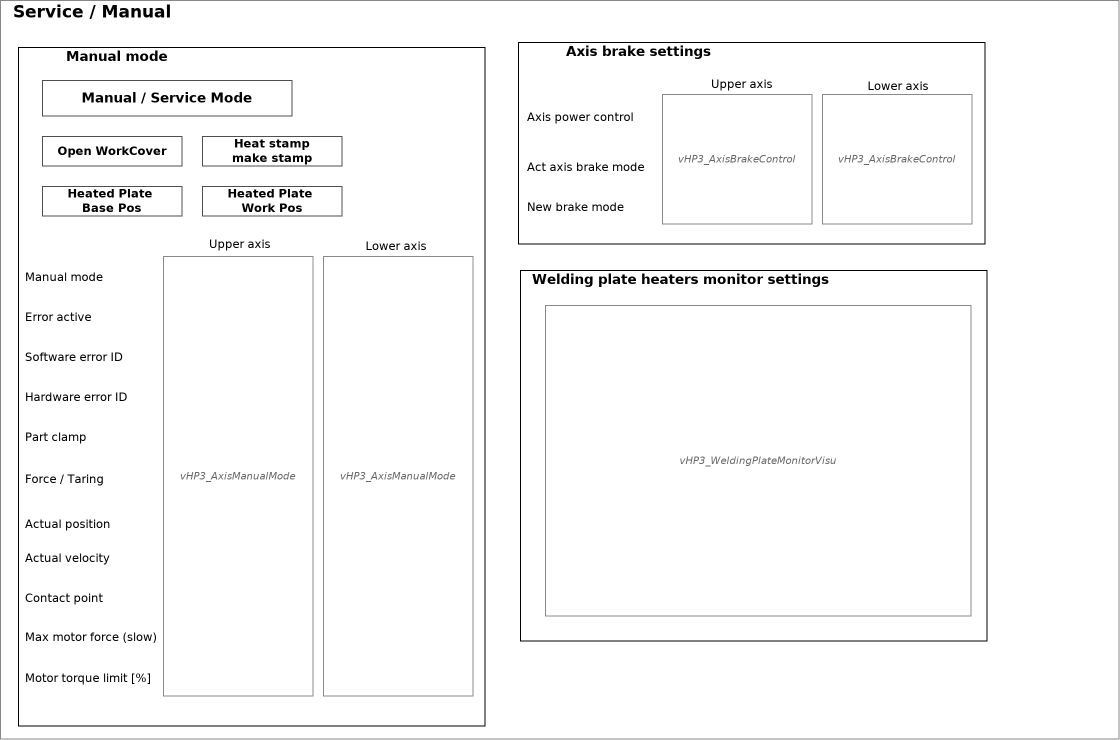
VISUALIZATION vHP3_MachineSub_Service  // 1120x740
VAR_IN_OUT
	fbHP: fbHPv3_Control;
END_VAR
    RoundedRectangle (18,47 467x679), "Manual mode"
    Rectangle (42,80 250x36), "Manual / Service Mode", colour toggle: fbHP.bManualMode
        toggle fbHP.bManualMode
    Label (22,265 130x24), "Manual mode"
    Label (22,512 130x24), "Actual position"
    Label (22,546 130x24), "Actual velocity"
    Label (22,625 145x24), "Max motor force (slow)"
    Rectangle (42,136 140x30), "Open WorkCover", colour toggle: fbHP.bWorkCover_Riseup, input disabled if: NOT fbHP.bManualMode
        toggle fbHP.bWorkCover_Riseup p2164770859=TRUE
    Rectangle (42,186 140x30), "Heated Plate Base Pos", colour toggle: fbHP.fbHeatedPlate_Actuator.Closed, input disabled if: NOT fbHP.bManualMode
        OnMouseClick: execute { fbHP.fbHeatedPlate_Actuator.mClose(); }
    Rectangle (202,186 140x30), "Heated Plate Work Pos", colour toggle: fbHP.fbHeatedPlate_Actuator.Opened, input disabled if: NOT fbHP.bManualMode
        OnMouseClick: execute { fbHP.fbHeatedPlate_Actuator.mOpen(); }
    Rectangle (202,136 140x30), "Heat stamp make stamp", colour toggle: fbHP.bMakeStamp, invisible if: NOT fbHP.bMarkingAsembled, input disabled if: NOT fbHP.bManualMode
        toggle fbHP.bMakeStamp
        OnMouseClick: execute { fbHP.fbHeatedPlate_Actuator.mClose(); }
    Label (175,232 130x24), "Upper axis"
    Label (331,234 130x24), "Lower axis"
    Label (22,666 145x24), "Motor torque limit [%]"
    RoundedRectangle (10,0 300x26), "Service / Manual"
    Frame (163,256 150x440)
        shows vHP3_AxisManualMode(fbData := fbHP.fbAxisUp)
    Frame (323,256 150x440)
        shows vHP3_AxisManualMode(fbData := fbHP.fbAxisDn)
    Label (22,305 130x24), "Error active"
    Label (22,345 130x24), "Software error ID"
    Label (22,385 130x24), "Hardware error ID"
    Label (22,467 130x24), "Force / Taring"
    Label (22,425 130x24), "Part clamp"
    Label (22,586 130x24), "Contact point"
    RoundedRectangle (518,42 467x202), "Axis brake settings"
    Label (524,105 130x24), "Axis power control"
    Label (677,72 130x24), "Upper axis"
    Label (833,74 130x24), "Lower axis"
    Label (524,155 130x24), "Act axis brake mode"
    Label (524,195 130x24), "New brake mode"
    Frame (662,94 150x130)
        shows vHP3_AxisBrakeControl(fbData := fbHP.fbAxisUp)
    Frame (822,94 150x130)
        shows vHP3_AxisBrakeControl(fbData := fbHP.fbAxisDn)
    RoundedRectangle (520,270 467x371), "Welding plate heaters monitor settings"
    Frame (545,305 426x311)
        shows vHP3_WeldingPlateMonitorVisu(fbData := fbHP.fbWeldingPlateHeaterChecker)
END_VISUALIZATION

(* stored: Version 1.1.0.1, ProductVersion 3.1.4024.15
   Visu vHP3_MachineSub_Service: Id {ff082b50-63b4-4d59-afc3-182679bbf1d2} *)
